(* PLC project Tc2_Utilities.F_SINT Demo, tc3-libraries-kb TwinCAT 3.1 *)
(* stored: creationDateTime 2026-05-11T00:00:00, modificationDateTime 2026-05-11T00:00:00 *)

PROGRAM P_Demo_F_SINT
  VAR
    nTempOffset : SINT := -12;  (* 业务量（SINT） *)
    bPackArg : BOOL;  (* 在线置 TRUE 触发一次打包 *)
    argDescriptor : T_Arg;  (* 打包后的 T_Arg 描述符（含 eType/cbLen/pData） *)
  END_VAR

            // ============================================================
// Tc2_Utilities.F_SINT 演示程序（FUNCTION，返回 T_Arg）
// ============================================================
// 场景：把 SINT 业务量打包为 T_Arg，供下游 EventLogger / FormatString2
//       / ADS 消息的可变参数机制使用。
// 价值：替代手填 T_Arg 三字段（eType/cbLen/pData），一行调用搞定。
// 验证：在线写 nTempOffset 为示例值，bPackArg := TRUE；
//       下一周期 argDescriptor.cbLen = SIZEOF(SINT)，argDescriptor.pData <> 0。
// ============================================================

IF bPackArg THEN
    // 单次完整调用：返回的 T_Arg 立即可喂给 F_PutInArg(arg := argDescriptor, ...)
    argDescriptor := F_SINT(nTempOffset);
    bPackArg := FALSE;
END_IF;

          
END_PROGRAM
